FUNCTION_BLOCK FB_RV_St_Zustandscheck
VAR_IN_OUT
	Zustand		: ST_RV_Zustand;
END_VAR
VAR_INPUT
END_VAR
VAR_OUTPUT
END_VAR
VAR
END_VAR

(*
	Stoerung_Code
		0:	Allgemein Störung Regelventil (intern)

	Warnung_Code
		0:	Allgemein Warnung Regelventil (intern)

*)
(* Interne Stoerungen / Warnungen *)


(* ------------------------------------------------------------------- *)
(* Stoermeldung *)
IF Zustand.Stoerung_Code > 0 THEN
	Zustand.Stoerung := TRUE;
(*ELSE - wird nur durch Quittierung gelöscht
	Zustand.Stoerung := FALSE; *)
END_IF;

(* Warnmeldung *)
IF Zustand.Warnung_Code > 0 THEN
	Zustand.Warnung := TRUE;
ELSE
	Zustand.Warnung := FALSE;
END_IF;

END_FUNCTION_BLOCK

(* stored: Version 1.1.0.1, ProductVersion 3.1.4024.9
   POU FB_RV_St_Zustandscheck: Id {4525baa4-67eb-4f0c-bb21-3cf0d3ea6342}, SpecialFunc None *)
